FUNCTION_BLOCK ChanSendBool (* Composite Function Block Type *)
  (* Standard: 61499-2 *)
  (* Version 0.0, 12/6/2023, vaatmar1, nxtControl GmBH, template *)
  PACKAGE Main;
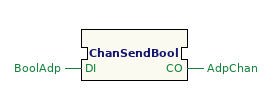
  SOCKETS
    DI : BoolAdp;
  END_SOCKETS
  PLUGS
    CO : AdpChan;
  END_PLUGS
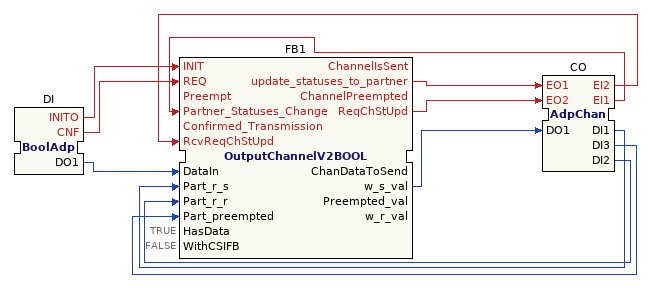
  FBS
    FB1 : OutputChannelV2BOOL(WithCSIFB := FALSE, HasData := TRUE);
  END_FBS
  EVENT_CONNECTIONS
    DI.INITO TO FB1.INIT;
    DI.CNF TO FB1.REQ;
    FB1.update_statuses_to_partner TO CO.EO1;
    FB1.ReqChStUpd TO CO.EO2;
    CO.EI2 TO FB1.RcvReqChStUpd;
    CO.EI1 TO FB1.Partner_Statuses_Change;
  END_CONNECTIONS
  DATA_CONNECTIONS
    FB1.w_s_val TO CO.DO1;
    DI.DO1 TO FB1.DataIn;
    CO.DI1 TO FB1.Part_r_s;
    CO.DI3 TO FB1.Part_preempted;
    CO.DI2 TO FB1.Part_r_r;
  END_CONNECTIONS
END_FUNCTION_BLOCK
